FUNCTION F_TargetReached : BOOL
VAR_INPUT
	fCurrentPos: LREAL;
	fTargetPos: LREAL;
END_VAR

F_TargetReached := F_TargetWindowReached(fCurrentPos, fTargetPos, fEpsilon);

END_FUNCTION

(* stored: Version 1.1.0.1, ProductVersion 3.1.4020.12
   POU F_TargetReached: Id {014ac5bc-4af5-4f8d-b06a-1aab6b15304e}, SpecialFunc None *)
